Universal Robots PolyScope program: groep3_robot_arm.urp

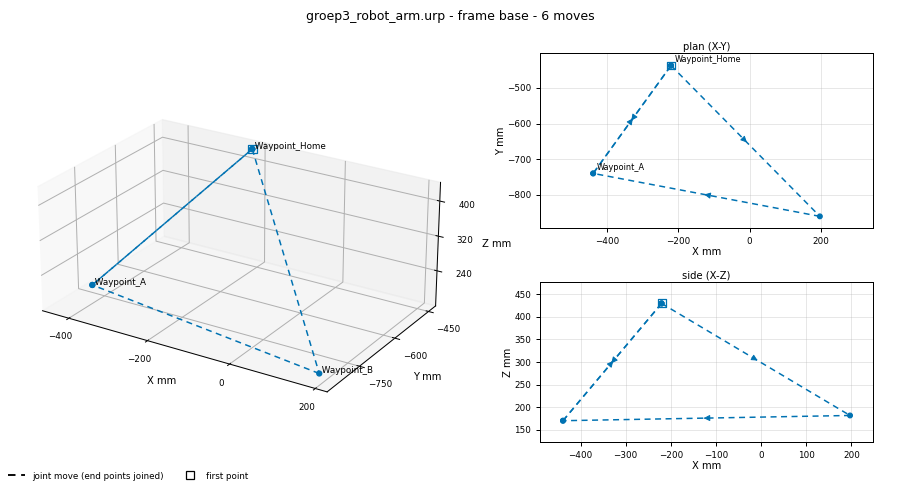
[picture p0: tool path of groep3_robot_arm.urp in frame base, 6 of 6 moves have a stored position in this frame; points joined in program order, loops and branches not executed]
Program groep3_robot_arm (installation=default directory=/home/ur/ursim-current/programs createdIn=3.15.6.106324 lastSavedIn=3.15.8.106339 robotSerialNumber=2018359999)
Calibrated DH parameters: a=[0.000173, -0.08184, -0.390569, 0.000014, 0.000061, 0]; d=[0.089465, 325.63058, -320.968373, -4.551618, 0.094907, 0.082699]; alpha=[1.570634, -0.001282, 0.007518, 1.570171, -1.57068, 0]; deltaTheta=[0.000011, -1.377212, 1.46664, -0.089508, -0.000013, 0.000027]
Robot Program (runOnlyOnce=false)
  If digital_in[4] == True
    MoveJ speed 60 deg/s, acceleration 80 deg/s^2 (useActiveTCP=true)
      Waypoint Waypoint_Home: TCP in base x=-220.525 y=-437.321 z=429.887 mm, rx=-1.0402 ry=-2.8991 rz=0.093 rad; joints [50.482, -92.028, 93.28, -95.659, -91.585, 0.009] deg
      Set SingleDigitalPulseActionState SingleDigitalPulseActionState(hiPulseInSeconds=0.5, pin=digital_out[4])
  Loop While (checkContinuously=false) expression=digital_in[4] == True
    If digital_in[6] == True
      Set IncrementVariable installationVariable=step_count
      If step_count > 2
        step_count := 0
      Switch expression=step_count
        Case (caseValue=1)
          MoveJ speed 60 deg/s, acceleration 80 deg/s^2 (useActiveTCP=true)
            Waypoint Waypoint_Home: TCP in base x=-220.525 y=-437.321 z=429.887 mm, rx=-1.0402 ry=-2.8991 rz=0.093 rad; joints [50.482, -92.028, 93.28, -95.659, -91.585, 0.009] deg
            Waypoint Waypoint_A: TCP in base x=-439.037 y=-740.017 z=170 mm, rx=-1.0074 ry=-2.9466 rz=-0.0457 rad; joints [52.227, -29.233, 35.48, -95.162, -92.018, -0.006] deg
        Case (caseValue=2)
          MoveJ speed 60 deg/s, acceleration 80 deg/s^2 (useActiveTCP=true)
            Waypoint Waypoint_Home: TCP in base x=-220.525 y=-437.321 z=429.887 mm, rx=-1.0402 ry=-2.8991 rz=0.093 rad; joints [50.482, -92.028, 93.28, -95.659, -91.585, 0.009] deg
            Waypoint Waypoint_B: TCP in base x=197.078 y=-860.501 z=181.621 mm, rx=0.1612 ry=-3.1032 rz=0.04 rad; joints [95.824, -24.35, 24.647, -91.658, -91.582, 0.008] deg
      Set SingleDigitalPulseActionState SingleDigitalPulseActionState(hiPulseInSeconds=0.5, pin=digital_out[4])
  MoveJ speed 60 deg/s, acceleration 80 deg/s^2 (useActiveTCP=true)
    Waypoint Waypoint_A: TCP in base x=-439.037 y=-740.017 z=170 mm, rx=-1.0074 ry=-2.9466 rz=-0.0457 rad; joints [52.227, -29.233, 35.48, -95.162, -92.018, -0.006] deg
    Set SingleDigitalPulseActionState SingleDigitalPulseActionState(hiPulseInSeconds=0.5, pin=digital_out[6])
    Halt
